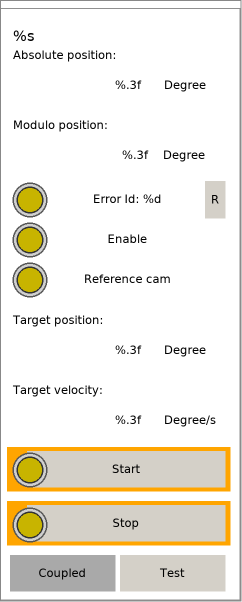
VISUALIZATION TplAxisControl  // 242x602
VAR_IN_OUT
	sAxisDescription				:STRING;
	fAbsolutePositon				:LREAL;
	fModuloPositon					:LREAL;
	bError							:BOOL;
	nErrorId						:DWORD;
	bReset							:BOOL;
	bPowerStatus					:BOOL;
	bReferenceCam					:BOOL;
	fMoveAbsPosition				:LREAL;
	fMoveAbsVelocity				:LREAL;
	bStartMoveAbs					:BOOL;
	bMoveAbsBusy					:BOOL;
	bMoveAbsDone					:BOOL;
	bStop							:BOOL;
	bStopBusy						:BOOL;
	bStopDone						:BOOL;
	bAxisCoupled					:BOOL;
	bTestChangeTargetPosAxis		:BOOL;
END_VAR
(* End *)
    GroupBox (0,0 240x600)
        Rectangle (7,501 223x44), invisible if: NOT bStopBusy
        Rectangle (7,447 223x44), invisible if: NOT bMoveAbsBusy
        Rectangle (27,451 198x36), "Start", colour toggle: bStartMoveAbs
            toggle bStartMoveAbs
        Group (10,110 230x60)
            Rectangle (0,30 148x30), "%.3f", text variable: fModuloPositon
            Label (150,30 80x30), "Degree"
            Label (0,0 200x30), "Modulo position:"
        Group (10,40 227x60)
            Rectangle (0,30 148x30), "%.3f", text variable: fAbsolutePositon
            Label (151,30 76x30), "Degree"
            Label (0,0 216x30), "Absolute position:"
        Group (10,180 200x40)
            Rectangle (20,1 195x36), "Error Id: %d", text variable: nErrorId
            Lamp1 (0,0 40x40), variable: bError, style: Lamp-Lamp1-Yellow
        Group (10,220 215x40)
            Rectangle (20,1 195x36), "Enable"
            Lamp1 (0,0 40x40), variable: bPowerStatus, style: Lamp-Lamp1-Yellow
        Group (10,260 215x40)
            Rectangle (20,1 195x36), "Reference cam"
            Lamp1 (0,0 40x40), variable: bReferenceCam, style: Lamp-Lamp1-Yellow
        Rectangle (205,181 20x37), "R", tooltip "Reset", colour toggle: bReset
            tap bReset
        Rectangle (27,505 198x36), "Stop", colour toggle: bStop
            toggle bStop
        Rectangle (10,555 105x36), "Coupled", colour toggle: bAxisCoupled
        Rectangle (10,25 230x22), "%s", text variable: sAxisDescription
        Rectangle (10,335 148x30), "%.3f", text variable: fMoveAbsPosition
            OnMouseClick: write the text variable via VisuDialogs.Numpad
        Label (161,335 76x30), "Degree"
        Label (10,305 216x30), "Target position:"
        Rectangle (10,405 148x30), "%.3f", text variable: fMoveAbsVelocity
            OnMouseClick: write the text variable via VisuDialogs.Numpad
        Label (161,405 76x30), "Degree/s"
        Label (10,375 216x30), "Target velocity:"
        Lamp1 (10,505 40x40), variable: bStopDone, style: Lamp-Lamp1-Yellow
        Rectangle (120,555 105x36), "Test", colour toggle: bTestChangeTargetPosAxis
            toggle bTestChangeTargetPosAxis
        Lamp1 (10,450 40x40), variable: bMoveAbsDone, style: Lamp-Lamp1-Yellow
END_VISUALIZATION

(* stored: Version 1.1.0.1, ProductVersion 3.1.4024.11
   Visu TplAxisControl: Id {35ad3630-b351-40af-9490-6cde31e24410} *)
